# EPICS IOC start-up script: require/3.1.2/siteMods/ess/0.0.1/iocLog.iocsh
#- ###               iocLog iocsh                   ###
#- ########################################$###########
#- >> Mandatory
#- IOCNAME        - IOC NAME
#- LOG_INET       - EPICS_IOC_LOG_INET
#- >> Optional
#- LOG_INET_PORT  - EPICS_IOC_LOG_PORT,  Default : 7004
#- LOGDISABLE     - log enalble,         Default : 0
#- FACNAME        - facility name,       Default :
#- #########################################$##########

epicsEnvSet(EPICS_IOC_LOG_INET, "$(LOG_INET)")
epicsEnvSet(EPICS_IOC_LOG_PORT, "$(LOG_INET_PORT=7004)")
epicsEnvSet(iocLogDisable, "$(LOGDISABLE=0)")
iocLogPrefix("fac=$(FACNAME=) proc=$(IOCNAME)");

# require has afterInit function
afterInit("iocLogInit()")
